// TIA Portal V20 export
DATA_BLOCK "IDB_HardwareDiag"   // DB12
// stored: Access Published, InstanceOfName Global.FB_HardwareDiag, InstanceOfType FB, Namespace Global
"Global.FB_HardwareDiag"
   // VAR
   //    "BW-ASi -10.106.129.143" : "Global.FB_GetDiag";
   //    "BW-ASi -10.106.129.200" { S7_SetPoint := 'True'} : "Global.FB_GetDiag";
   //    "Cognex -10.106.129.24" : "Global.FB_GetDiag";
   //    "Cognex -10.106.129.25" { S7_SetPoint := 'True'} : "Global.FB_GetDiag";
   //    "Cognex -10.106.129.26" { S7_SetPoint := 'True'} : "Global.FB_GetDiag";
   //    "Cognex -10.106.129.27" { S7_SetPoint := 'True'} : "Global.FB_GetDiag";
   //    "IMC - 10.106.129.84" { S7_SetPoint := 'True'} : "Global.FB_GetDiag";
   //    "IMC - 10.106.129.85" { S7_SetPoint := 'True'} : "Global.FB_GetDiag";
   //    "IMC - 10.106.129.86" { S7_SetPoint := 'True'} : "Global.FB_GetDiag";
   //    "IMC - 10.106.129.87" { S7_SetPoint := 'True'} : "Global.FB_GetDiag";
   //    "IMC - 10.106.129.88" { S7_SetPoint := 'True'} : "Global.FB_GetDiag";
   // END_VAR
BEGIN
END_DATA_BLOCK
